// TIA Portal V19 export
ORGANIZATION_BLOCK "Startup"   // OB3030, LAD, Startup
TITLE = "Complete Restart"
AUTHOR : Siemens_FA_SUP
// stored: AutoNumber false, IsIECCheckEnabled true, Namespace Unit.Em2, SetENOAutomatically true
   VAR_INPUT
      LostRetentive : Bool;   // True if retentive data are lost
      LostRTC : Bool;   // True if date and time are lost
   END_VAR
BEGIN

REGION Network 1 (SCL): Build the Absolut Reference Designator
   // Set the Absoult Reference Designator in the Config DB
   IF LEN(IN := "Unit.Em2.Config".em.referenceDesignator.parent) <> 0 THEN
       "Unit.Em2.Config".em.referenceDesignator.combined := CONCAT_WSTRING(IN1 := "Unit.Em2.Config".em.referenceDesignator.parent, IN2 := WSTRING#'.', IN3 := "Unit.Em2.Config".em.referenceDesignator.relative);
   ELSE
       "Unit.Em2.Config".em.referenceDesignator.combined := "Unit.Em2.Config".em.referenceDesignator.relative;
   END_IF;
END_REGION

REGION Network 2 (SCL): Axes data
   // Assign axes
   "Unit.Em2.Config".axis[1] := "Em2_PositioningAxis";
   "Unit.Em2.Config".axis[2] := "Em2_SynchronousAxis";
END_REGION
END_ORGANIZATION_BLOCK
